# B&R Automation Studio project NAINV104C00R8L515F00 (part 38)

#### Act_OpsRun.st
```iecst
(** 2019-03-25 **)
ACTION Act_OpsRun:

	IF eSimuInvGotoStep	<> eSimuInvStep THEN
		CASE eSimuInvGotoStep OF

			ELSE
				fbInvChgDirDlyTm(IN := FALSE);
				fbConvChgDirDlyTm(IN := FALSE);
				eSimuInvStep	:= eSimuInvGotoStep;
		END_CASE

	END_IF

	IF eSimuInvGotoStep = eSimuInvStep THEN

		IF bPaused = FALSE THEN

			CASE eSimuInvStep OF

				SimuInvStepChkCondition :

					IF p_bInletShutterCloseRs = FALSE OR p_bOutletShutterCloseRs = FALSE THEN
						eSimuInvGotoStep := SimuInvStepInitShutterCls;

					ELSE
						IF p_bStopperExtended = FALSE THEN
							eSimuInvGotoStep	:= SimuInvStepInitStopperExt;
						END_IF

					END_IF

					bPaused	 := p_bStop OR p_bStep;

				SimuInvStepInitShutterCls:

					eInShutterAct 	:= PneuActExt;
					eOutShutterAct	:= PneuActExt;

					IF (p_eInletShutterStat = PneuActExt AND p_eInletShutterStatus = Done) AND (p_eOutletShutterStat = PneuActExt AND p_eOutletShutterStatus = Done) THEN

						eInShutterAct := PneuActIdle;
						eOutShutterAct := PneuActIdle;

						eSimuInvGotoStep := SimuInvStepInitStopperExt;

						bPaused	:= p_bStop OR p_bStep;

					END_IF

				SimuInvStepInitStopperExt:

					eStopperAct	:= PneuActExt;

					IF (p_eStopperStat = PneuActExt AND p_eStopperStatus = Done) THEN

						eStopperAct	 := PneuActIdle;

						IF  p_bInverterHomeSen AND p_bConvRightSen THEN
							eSimuInvGotoStep	:= SimuInvStepInvertRemote;

						ELSIF p_bInverterHomeSen AND (p_bConvLeftSen OR NOT (p_bConvLeftSen OR p_bConvRightSen) ) THEN
							eSimuInvGotoStep 	:= SimuInvStepConvToRightSen;

						ELSIF p_bInverterRemoteSen AND p_bConvLeftSen THEN
							eSimuInvGotoStep	:= SimuInvStepInvertHome;

						ELSIF p_bInverterRemoteSen AND (p_bConvRightSen OR NOT (p_bConvLeftSen OR p_bConvRightSen) ) THEN
							eSimuInvGotoStep	:= SimuInvStepConvToLeftSen;

						ELSIF NOT(p_bInverterHomeSen OR p_bInverterRemoteSen) THEN
							eSimuInvGotoStep	:= SimuInvStepInvertHome;

						END_IF

						bPaused	:= p_bStop OR p_bStep;

					END_IF

				SimuInvStepInvertHome:

					eInverterAct := MotorBrkActCCW;

					IF (p_eInvertStat = MotorBrkActCCW AND p_eInvertStatus = Done) THEN

						eInverterAct 	:= MotorBrkActIdle;

						fbInvChgDirDlyTm(IN := TRUE);

						IF fbInvChgDirDlyTm.Q THEN //After Inverter invert to Home postion and time up the Waiting Time , Board go to conv Exit sensor

							eConvAct := ConvActEnt;
							fbInvChgDirDlyTm(IN := FALSE);

							IF (p_eConvStat = ConvActEnt AND p_eConvStatus = Done) THEN
								fbConvChgDirDlyTm (IN := TRUE);
							END_IF

						END_IF

						IF fbConvChgDirDlyTm.Q THEN // Board reach the Conv Exit sensor and time up the Waiting Time , Board go back to the conv Inlet sensor

							eConvAct	:= ConvActRev;
							fbConvChgDirDlyTm(IN := FALSE);

							IF (p_eConvStat = ConvActRev AND p_eConvStatus = Done) THEN // Board Reach the conv Inlet sensor, will go back to conv Exit sensor
								eConvAct	:= ConvActRevImmedStart;
							END_IF
						END_IF

						IF p_ConvStat = ConvActRevImmedStart AND p_eConvStatus = Done THEN

							eConvAct	:= ConvActIdle;

							fbInvChgDirDlyTm(IN := TRUE);

							IF fbInvChgDirDlyTm.Q THEN // Board Reach the conv Exit sensor and time up the Waiting Time, Inverter will start Invert to Remote Position
								eSimuInvGotoStep	:= SimuInvStepInvertRemote;
								fbInvChgDirDlyTm(IN := FALSE);
							END_IF

						END_IF

						bPaused	:= p_bStop OR p_bStep;

					END_IF

				SimuInvStepInvertRemote:

					eInverterAct	:= MotorBrkActCW;

					IF (p_eInvertStat = MotorBrkActCW AND p_eInvertStatus = Done) THEN

						eInverterAct	:= MotorBrkActIdle;

						fbInvChgDirDlyTm(IN := TRUE);

						IF fbInvChgDirDlyTm.Q THEN

							eConvAct	:=  ConvActEnt;
							fbInvChgDirDlyTm(IN := FALSE);

							IF p_eConvStat= ConvActEnt AND p_eConvStatus = Done THEN
								fbConvChgDirDlyTm (IN := TRUE);
							END_IF

							IF fbConvChgDirDlyTm.Q THEN
								fbConvChgDirDlyTm (IN := FALSE);
								eConvAct	:= ConvActRev;
							END_IF

							IF p_eConvStat = ConvActRev AND p_eConvStatus = Done THEN
								eConvAct	:= ConvActIdle;
								fbInvChgDirDlyTm (IN := TRUE);
							END_IF

							IF fbInvChgDirDlyTm.Q THEN
								eSimuInvGotoStep := SimuInvStepInvertHome;
								fbInvChgDirDlyTm (IN:= FALSE);

							END_IF

						END_IF

						bPaused	:= p_bStop OR p_bStep;

					END_IF

				SimuInvStepConvToRightSen:

					eConvAct	:= ConvActInit;

					IF (p_eConvStat = ConvActInit AND p_eConvStatus = Done) THEN

						eConvAct :=	ConvActIdle;

						eSimuInvGotoStep	:= SimuInvStepInvertRemote;

						bPaused := p_bStop OR p_bStep;

					END_IF

				SimuInvStepConvToLeftSen:

					eConvAct	:= ConvActRev;

					IF (p_eConvStat = ConvActRev AND p_eConvStatus = Done) THEN

						eConvAct	:= ConvActIdle;

						eSimuInvGotoStep	:= SimuInvStepInvertHome;

						bPaused := p_bStop OR p_bStep;

					END_IF

			END_CASE

		END_IF

	END_IF

END_ACTION
```

#### Act_OpsRst.st - Do Not Change!!!
```iecst
(** 2019-03-25 **)
ACTION Act_OpsRst:

	eInverterAct			:= MotorBrkActIdle;
	eConvAct				:= ConvActIdle;
	eInShutterAct			:= PneuActIdle;
	eOutShutterAct			:= PneuActIdle;
	eStopperAct				:= PneuActIdle;

	fbInvChgDirDlyTm(IN:=FALSE);
	fbConvChgDirDlyTm(IN:=FALSE);

END_ACTION
```

#### InputRef.var - Do Not Change!!!
```iecst
(*2019-03-25*)
(**)
(*General*)
VAR
	p_udiRstErr : REFERENCE TO UDINT;
	p_bEn : REFERENCE TO BOOL;
	p_bDis : REFERENCE TO BOOL;
	p_bRun : REFERENCE TO BOOL;
	p_bStop : REFERENCE TO BOOL;
	p_bStep : REFERENCE TO BOOL;
END_VAR
(**)
VAR
	p_bInletShutterPrep : REFERENCE TO BOOL;
	p_bOutletShutterPrep : REFERENCE TO BOOL;
END_VAR
(**)
VAR
	p_sProgNm : REFERENCE TO STRING[15];
	p_bNtSettingsLoadDone : REFERENCE TO BOOL;
END_VAR
(**)
VAR
	p_eInvertStat : REFERENCE TO eMotorBrkAction;
	p_eInvertStatus : REFERENCE TO eFBStatus;
	p_eConvStat : REFERENCE TO eConvAction;
	p_eConvStatus : REFERENCE TO eFBStatus;
	p_eStopperStat : REFERENCE TO ePneuAction;
	p_eStopperStatus : REFERENCE TO eFBStatus;
	p_eInletShutterStat : REFERENCE TO ePneuAction;
	p_eInletShutterStatus : REFERENCE TO eFBStatus;
	p_eOutletShutterStat : REFERENCE TO ePneuAction;
	p_eOutletShutterStatus : REFERENCE TO eFBStatus;
END_VAR
(**)
VAR
	p_bConvLeftSen : REFERENCE TO BOOL;
	p_bConvRightSen : REFERENCE TO BOOL;
	p_bInverterHomeSen : REFERENCE TO BOOL;
	p_bInverterRemoteSen : REFERENCE TO BOOL;
	p_bStopperExtended : REFERENCE TO BOOL;
	p_bStopperRetracted : REFERENCE TO BOOL;
	p_bInletShutterOpenRs : REFERENCE TO BOOL;
	p_bInletShutterCloseRs : REFERENCE TO BOOL;
	p_bOutletShutterOpenRs : REFERENCE TO BOOL;
	p_bOutletShutterCloseRs : REFERENCE TO BOOL;
END_VAR
```

#### Local.var - Do Not Change!!!
```iecst
(*2019-03-25*)
(**)
(*Local Action, State & Status*)
VAR
	eStatus : eFBStatus := Idle;
	udiStatus : UDINT := 0;
END_VAR
(**)
(*Local Alarm*)
VAR
	tyAlmData : tyAlmDat;
	a_tyAlmText : ARRAY[10000..10099] OF tyAlmTxt;
END_VAR
(**)
(*Local Output*)
VAR
	sStepTxt : STRING[80];
	bPaused : BOOL;
	eInverterAct : eMotorBrkAction;
	eConvAct : eConvAction;
	eInShutterAct : ePneuAction;
	eOutShutterAct : ePneuAction;
	eStopperAct : ePneuAction;
END_VAR
(**)
(*Local Input*)
VAR
	udiRstErr : UDINT := 0;
	bEn : BOOL := TRUE;
	bDis : BOOL := FALSE;
	bRun : BOOL;
	bStop : BOOL;
	bStep : BOOL;
END_VAR
(**)
VAR
	bInvHomeSen : BOOL;
	binvRemoteSen : BOOL;
	bConvLeftSen : BOOL;
	bConvRightSen : BOOL;
	bInletShutterCloseRS : BOOL;
	bOutletShutterCloseRS : BOOL;
END_VAR
(**)
VAR
	eInverterStat : eMotorBrkAction;
	eInverterStatus : eFBStatus;
	eConvStat : eConvAction;
	eConvStatus : eFBStatus;
	eInletShutterStat : ePneuAction;
	eInletShutterStatus : eFBStatus;
	eOutletShutterStat : ePneuAction;
	eOutletShutterStatus : eFBStatus;
	eStopperStat : ePneuAction;
	eStopperStatus : eFBStatus;
END_VAR
(**)
VAR
	sProgNm : STRING[15];
	bNtSettingsLoadDone : BOOL := TRUE;
END_VAR
(**)
(*Local*)
VAR
	bRstErr : BOOL;
	udiRstErrOld : UDINT;
	bInitDone : BOOL;
	bInitialDone : BOOL;
	eSimuInvStep : eSimuInvRunStep := SimuInvStepNA;
	eSimuInvGotoStep : eSimuInvRunStep := SimuInvStepChkCondition;
	fbInvChgDirDlyTm : TON := (PT:=T#5s);
	fbConvChgDirDlyTm : TON := (PT:=T#5s);
END_VAR
```

Listed in the project but not available here: Logical/UI/UI/Act_LinkAction.st, Logical/UI/UI/Act_Background/Action/C0001, Logical/UI/UI/Act_Background/Action/C0002, Logical/UI/UI/Act_Background/Action/C0003, Logical/UI/UI/Act_Background/Action/C0006, Logical/Startup/Startup/Act_LinkAction.st, Logical/UsrFolder/UsrFolder/Act_Link.st, Logical/UsrFolder/UsrFolder/Act_RstErr.st, Logical/Time/Time/InputRef_Link.var, Logical/Time/Time/Act_LinkAction.st, Logical/Time/Time/Act_Link.st, Logical/Time/Time/Act_RstErr.st, Logical/RstErr/RstErr/Act_Link.st, Logical/RstErr/RstErr/Cyclic.st, Logical/ProdRcp/ProdRcp/Act_RstErr.st, Logical/SMEMA/USSMEMA/Act_LinkEn.st, Logical/SMEMA/USSMEMA/Cyclic.st, Logical/SMEMA/USSMEMA/Act_RstErr.st, Logical/SMEMA/USSMEMA/Act_Action.st, Logical/SMEMA/USSMEMA/Act_Main.st, Logical/SMEMA/USSMEMA/Act_Alarm.st, Logical/SMEMA/USSMEMA2/Act_LinkEn.st, Logical/SMEMA/USSMEMA2/Act_InitLocal.st, Logical/SMEMA/USSMEMA2/Act_Initial.st, Logical/SMEMA/USSMEMA2/Act_Background.st, Logical/SMEMA/USSMEMA2/InputRef.var, Logical/Pneu/PneuNoSenStopper/InputRef_Link.var, Logical/Pneu/PneuNoSenStopper/Act_LinkEn.st, Logical/Pneu/PneuNoSenStopper/Act_Link.st, Logical/Pneu/PneuNoSenStopper/Cyclic.st, Logical/Pneu/PneuNoSenStopper/Act_RstErr.st, Logical/Pneu/PneuNoSenStopper/Act_Action.st, Logical/Pneu/PneuNoSenStopper/Act_Main.st, Logical/Pneu/Pneu2SenInShutter/Act_LinkEn.st, Logical/Pneu/Pneu2SenInShutter/Act_Link.st, Logical/Pneu/Pneu2SenInShutter/Cyclic.st, Logical/Pneu/Pneu2SenInShutter/Act_RstErr.st, Logical/Pneu/Pneu2SenInShutter/Act_Action.st, Logical/Pneu/Pneu2SenInShutter/Act_Main.st, Logical/Pneu/Pneu2SenInShutter/InputRef.var, Logical/CANOpenServo/AW/AWOpen/Act_LinkEn.st, Logical/DOutput/DOutput/Act_Initial.st, Logical/Hermes/Hermes/Act_Action.st, Logical/Hermes/USHermes/Act_LinkAction.st, Logical/Hermes/USHermes/Act_Initial.st, Logical/Hermes/USHermes/Act_Background.st, Logical/Hermes/USHermes/Act_Background_Info.st, Logical/Hermes/USHermes/Act_Background_CmpParamRcv.st, Logical/Hermes/USHermes/Act_Background_BoardAvailableChk.st, Logical/Hermes/USHermes/Act_Background_ChkAlive.st, Logical/Hermes/USHermes/Act_Background_ChgConfig.st, Logical/Hermes/USHermes/Act_Background_ProcessData.st, Logical/Hermes/USHermes/Act_Background_TCPClose.st, Logical/Hermes/USHermes/Act_Background_Stop.st, Logical/Hermes/USHermes/Act_Background_Log.st, Logical/Hermes/USHermes/Act_Background_AccData.st, Logical/Hermes/USHermes/Act_Background_BFAccData.st, Logical/Hermes/USHermes/Act_Main_Disable.st, Logical/Hermes/USHermes/Act_CombineErr.st, Logical/Hermes/USHermes/Act_Alarm1.st, Logical/Hermes/USHermes/Act_Alarm5.st, Logical/Hermes/USHermes/InputRef.var, Logical/Hermes/USHermes/Act_Background_RequestedBoardChk.st, Logical/Hermes/DSHermes/Act_LinkEn.st, Logical/Hermes/DSHermes/Act_RstErr.st, Logical/Hermes/DSHermes/Act_Initial.st, Logical/Hermes/DSHermes/Act_Action.st, Logical/Hermes/DSHermes/Act_Main.st, Logical/Hermes/DSHermes/Act_Background_NotificationRcv.st, Logical/Hermes/DSHermes/Act_Background_IllegalMsg.st, Logical/Hermes/DSHermes/Act_Background_CmpParamRcv.st, Logical/Hermes/DSHermes/Act_Background_SequenceTO.st, Logical/Hermes/DSHermes/Act_Background_ChkAlive.st, Logical/Hermes/DSHermes/Act_Background_ChgConfig.st, Logical/Hermes/DSHermes/Act_Background_Command.st, Logical/Hermes/DSHermes/Act_Background_NotificationSnd.st, Logical/Hermes/DSHermes/Act_Background_TCPSend.st, Logical/Hermes/DSHermes/Act_Background_TCPCloseSvr.st, Logical/Hermes/DSHermes/Act_Background_Log.st, Logical/Hermes/DSHermes/Act_Background_Err.st, Logical/Hermes/DSHermes/Act_CombineErr.st, Logical/Hermes/DSHermes/Act_Alarm.st, Logical/Hermes/DSHermes/Act_Alarm1.st, Logical/Hermes/RmtHermes/Act_Background_Log.st, Logical/Hermes/RmtHermes/Act_CombineErr.st, Logical/Hermes/SvyHermes/Act_LinkEn.st, Logical/Hermes/SvyHermes/Act_RstErr.st, Logical/Hermes/SvyHermes/Act_Action.st, Logical/Hermes/SvyHermes/Act_Background_NotificationRcv.st, Logical/Hermes/SvyHermes/Act_Background_ChkAliveSendPing.st, Logical/Hermes/SvyHermes/Act_Background_ChkAliveRcvPing.st, Logical/Hermes/SvyHermes/Act_Background_Stop.st, Logical/LF/Follower1/Cyclic.st, Logical/LF/Follower1/Act_Initial.st, Logical/LF/Follower1/Act_Background_UpdtData.st, Logical/LF/Follower1/Act_Main_Disable.st, Logical/LCS/LCSMngRcp/Act_LinkAction.st, Logical/LCS/LCSMngRcp/Act_RstErr.st, Logical/LCS/LCSMngRcp/Act_Main_Disable.st, Logical/Operations/Ops/Act_LinkAction.st, Logical/Operations/Ops/Act_RstErr.st, Logical/Operations/Ops/Act_InitLocal.st, Logical/Operations/Ops/Act_Initial.st, Logical/Operations/OpsInvert/Act_Initial.st, Logical/Machine/Machine/Act_RstErr.st, Logical/MotorBrk/MotorBrk/Act_LinkEn.st, Logical/MotorBrk/MotorBrk/Act_RstErr.st, Logical/Simulation/Simu/Cyclic.st, Logical/Simulation/Simu/Act_RstErr.st, Logical/Simulation/SimuInv/Act_LinkEn.st, Logical/Simulation/SimuInv/Act_RstErr.st
